FUNCTION F_LinSens	:	ST_InputVar
VAR_INPUT
	stInput	:	ST_InputVar;
END_VAR
VAR
END_VAR

stInput.fVal	:=	stInput.fParaM * DINT_TO_REAL(stInput.nVarInput) + stInput.fParaC; //linear conversion

IF stInput.bSensErr THEN
	stInput.bValid	:=	FALSE;
END_IF

//check if value is valid
IF (stInput.fVal > stInput.fParaMaxVal) OR (stInput.fVal < stInput.fParaMinVal) THEN
	stInput.bValid	:=	FALSE;
END_IF

F_LinSens	:=	stInput;	//return

END_FUNCTION

(* stored: Version 1.1.0.1, ProductVersion 3.1.4018.2
   POU F_LinSens: Id {93407fe1-99d7-48bd-92cd-924237ac1e19}, SpecialFunc None *)
